TYPE
    ExampleCylinderConfig :
    STRUCT
        TimeToReachHomePosition : TIME := T#10S;
        TimeToReachWorkPosition : TIME := T#10S;
    END_STRUCT
END_TYPE

(* stored: Version 1.1.0.1, ProductVersion 3.1.4024.12
   DUT ExampleCylinderConfig: Id {2da9610d-8fa5-47ef-9ed7-863f4fa2f81e} *)
